TYPE ST_PMLControl_Simplified :
STRUCT
	bConfirmation			: BOOL;
	
	bClearEnabled			: BOOL;
	bResetEnabled			: BOOL;
	bStartEnabled			: BOOL;
	bStopEnabled			: BOOL;
	
	bClearPressed			: BOOL;
	bResetPressed			: BOOL;
	bStartPressed			: BOOL;
	bStopPressed			: BOOL;
END_STRUCT
END_TYPE

(* stored: Version 1.1.0.1, ProductVersion 3.1.4024.9
   DUT ST_PMLControl_Simplified: Id {8b696aa5-3c11-4027-9a46-563f5114abac} *)
